{attribute 'qualified_only'}
{attribute 'strict'}
TYPE E_MbErrorClass :
(
	None := 0,
	Timeout,
	Crc,
	Exception,
	Transport,
	Config,
	Truncated,
	StillFailing,
	Recovered
);
END_TYPE

(* stored: Version 1.1.0.1
   DUT E_MbErrorClass: Id {ba77ce8c-449b-4577-a0a4-517118165deb} *)
